_CFC_ (* Continuous Function Chart, elements in execution order *)
#0 WORD_TO_REAL(RD_2[0])
#1 DIV(#0, 100)
#2 SCHU_P2_1_M2_OBR <= #1
#3 dost_ton_2:TON(IN: NOT SCHU_P2_1_M2_OBR_ERROR, PT: t#10s)
#4 SR_DOST_M2:RS(SET: #3.Q, RESET1: SCHU_P2_1_M2_OBR_ERROR)
#5 fb_M2b30:ISTOK_GT(dost: #4.Q1, x: SCHU_P2_1_M2_OBR, ust: #14, shkal: -, gist: 1)
#6 SCHU_P2_1_M2_B30 <= #5.Xb
#7 fb_M2_OBRb45:ISTOK_GT(dost: #4.Q1, x: SCHU_P2_1_M2_OBR, ust: #16, shkal: -, gist: 1)
#8 SCHU_P2_1_M2_B45 <= #7.Xb
#9 fb_M2_OBRm0_1:ISTOK_LT(dost: #4.Q1, x: SCHU_P2_1_M2_OBR, ust: 0.1, shkal: -, gist: 1)
#10 SCHU_P2_1_M2_M0_1 <= #9.Xm
#11 fb_M2_OBRbSM:ISTOK_GT(dost: #4.Q1, x: SCHU_P2_1_M2_OBR, ust: SCHU_P2_1_M_MAXSPEED, shkal: -, gist: 1)
#12 SCHU_P2_1_M2_OBRBSM <= #11.Xb
(* 60% от частоты вращения *)
#13 DIV(SCHU_P2_1_M_MAXSPEED, 100)
#14 MUL(#13, 60)
#15 DIV(SCHU_P2_1_M_MAXSPEED, 100)
#16 MUL(#15, 85)
(* 85% от частоты вращения *)
_END_CFC_
END_PROGRAM

(* POU TZBiS/S/ALL_S, CFC *)
PROGRAM ALL_S
VAR
END_VAR
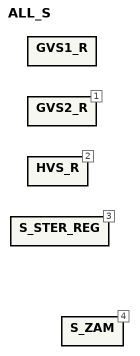
_CFC_ (* Continuous Function Chart, elements in execution order *)
#0 GVS1_R()
#1 GVS2_R()
#2 HVS_R()
#3 S_STER_REG()
#4 S_ZAM()
_END_CFC_
(* the same logic as Structured Text *)
GVS1_R();
GVS2_R();
HVS_R();
S_STER_REG();
S_ZAM();
END_PROGRAM

(* POU TZBiS/S/GVS1_R, CFC *)
PROGRAM GVS1_R
VAR
	rs_gvs1: RS;
	GVS1_RUN: BOOL;
END_VAR
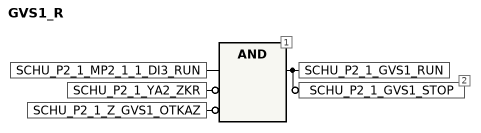
_CFC_ (* Continuous Function Chart, elements in execution order *)
#0 SCHU_P2_1_GVS1_RUN <= #1
#1 AND(SCHU_P2_1_MP2_1_1_DI3_RUN, NOT SCHU_P2_1_YA2_ZKR, NOT SCHU_P2_1_Z_GVS1_OTKAZ)
#2 SCHU_P2_1_GVS1_STOP <= NOT #1
_END_CFC_
END_PROGRAM

(* POU TZBiS/S/GVS2_R, CFC *)
PROGRAM GVS2_R
VAR
END_VAR
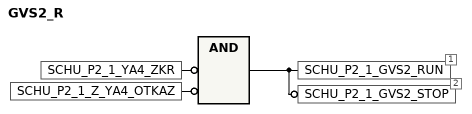
_CFC_ (* Continuous Function Chart, elements in execution order *)
#0 AND(NOT SCHU_P2_1_YA4_ZKR, NOT SCHU_P2_1_Z_YA4_OTKAZ)
#1 SCHU_P2_1_GVS2_RUN <= #0
#2 SCHU_P2_1_GVS2_STOP <= NOT #0
_END_CFC_
END_PROGRAM

(* POU TZBiS/S/HVS_R, CFC *)
PROGRAM HVS_R
VAR
END_VAR
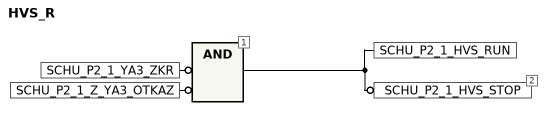
_CFC_ (* Continuous Function Chart, elements in execution order *)
#0 SCHU_P2_1_HVS_RUN <= #1
#1 AND(NOT SCHU_P2_1_YA3_ZKR, NOT SCHU_P2_1_Z_YA3_OTKAZ)
#2 SCHU_P2_1_HVS_STOP <= NOT #1
_END_CFC_
END_PROGRAM

(* POU TZBiS/S/S_STER_REG, CFC *)
PROGRAM S_STER_REG
VAR
	ZAD_S_Ster_Reg: TON;
END_VAR
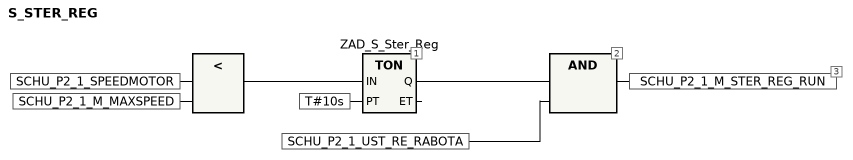
_CFC_ (* Continuous Function Chart, elements in execution order *)
#0 <(SCHU_P2_1_SPEEDMOTOR, SCHU_P2_1_M_MAXSPEED)
#1 ZAD_S_Ster_Reg:TON(IN: #0, PT: T#10s)
#2 AND(#1.Q, SCHU_P2_1_UST_RE_RABOTA)
#3 SCHU_P2_1_M_STER_REG_RUN <= #2
_END_CFC_
END_PROGRAM

(* POU TZBiS/S/S_ZAM, CFC *)
PROGRAM S_ZAM
VAR
	SR_ZAM: SR;
END_VAR
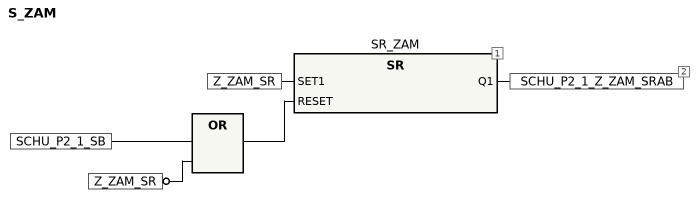
_CFC_ (* Continuous Function Chart, elements in execution order *)
#0 OR(SCHU_P2_1_SB, NOT Z_ZAM_SR)
#1 SR_ZAM:SR(SET1: Z_ZAM_SR, RESET: #0)
#2 SCHU_P2_1_Z_ZAM_SRAB <= #1.Q1
_END_CFC_
(* the same logic as Structured Text *)
SR_ZAM(SET1 := Z_ZAM_SR, RESET := SCHU_P2_1_SB OR NOT Z_ZAM_SR);
SCHU_P2_1_Z_ZAM_SRAB := SR_ZAM.Q1;
END_PROGRAM

(* POU TZBiS/TZB/ALL_TZB, CFC *)
PROGRAM ALL_TZB
VAR
END_VAR
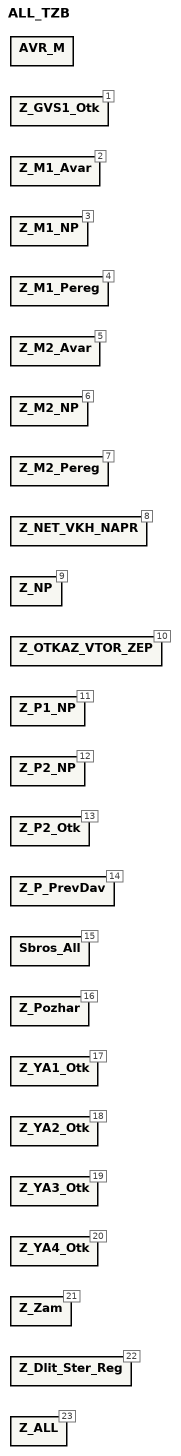
_CFC_ (* Continuous Function Chart, elements in execution order *)
#0 AVR_M()
#1 Z_GVS1_Otk()
#2 Z_M1_Avar()
#3 Z_M1_NP()
#4 Z_M1_Pereg()
#5 Z_M2_Avar()
#6 Z_M2_NP()
#7 Z_M2_Pereg()
#8 Z_NET_VKH_NAPR()
#9 Z_NP()
#10 Z_OTKAZ_VTOR_ZEP()
#11 Z_P1_NP()
#12 Z_P2_NP()
#13 Z_P2_Otk()
#14 Z_P_PrevDav()
#15 Sbros_All()
#16 Z_Pozhar()
#17 Z_YA1_Otk()
#18 Z_YA2_Otk()
#19 Z_YA3_Otk()
#20 Z_YA4_Otk()
#21 Z_Zam()
#22 Z_Dlit_Ster_Reg()
#23 Z_ALL()
_END_CFC_
(* the same logic as Structured Text *)
AVR_M();
Z_GVS1_Otk();
Z_M1_Avar();
Z_M1_NP();
Z_M1_Pereg();
Z_M2_Avar();
Z_M2_NP();
Z_M2_Pereg();
Z_NET_VKH_NAPR();
Z_NP();
Z_OTKAZ_VTOR_ZEP();
Z_P1_NP();
Z_P2_NP();
Z_P2_Otk();
Z_P_PrevDav();
Sbros_All();
Z_Pozhar();
Z_YA1_Otk();
Z_YA2_Otk();
Z_YA3_Otk();
Z_YA4_Otk();
Z_Zam();
Z_Dlit_Ster_Reg();
Z_ALL();
END_PROGRAM

(* POU TZBiS/TZB/AVR_M, CFC *)
PROGRAM AVR_M
VAR
	fb_HVACRC: FB_HVACRedundancyCtrl;
	RS_Pusk: RS;
	RT_Pusk: R_TRIG;


	rHours: ARRAY[1..8] OF REAL;
	uiCount: ARRAY[1..8] OF UINT;

	delayFBC: TIME := T#1s;
	overlap1Actuator: TIME := T#0s;
	maxOnLevel: UINT := 999;

	dtSystemTime: DT;
	fb_HVAC_GST: FB_HVACGetSystemTime;
	error: BOOL;
	RS_avr_kom: RS;
	RT_T: R_TRIG;
	TON_VKL: TON;
	TON_PUSK: TON;
	SCHU_P2_1_SA2_DI3_A: BOOL;
END_VAR
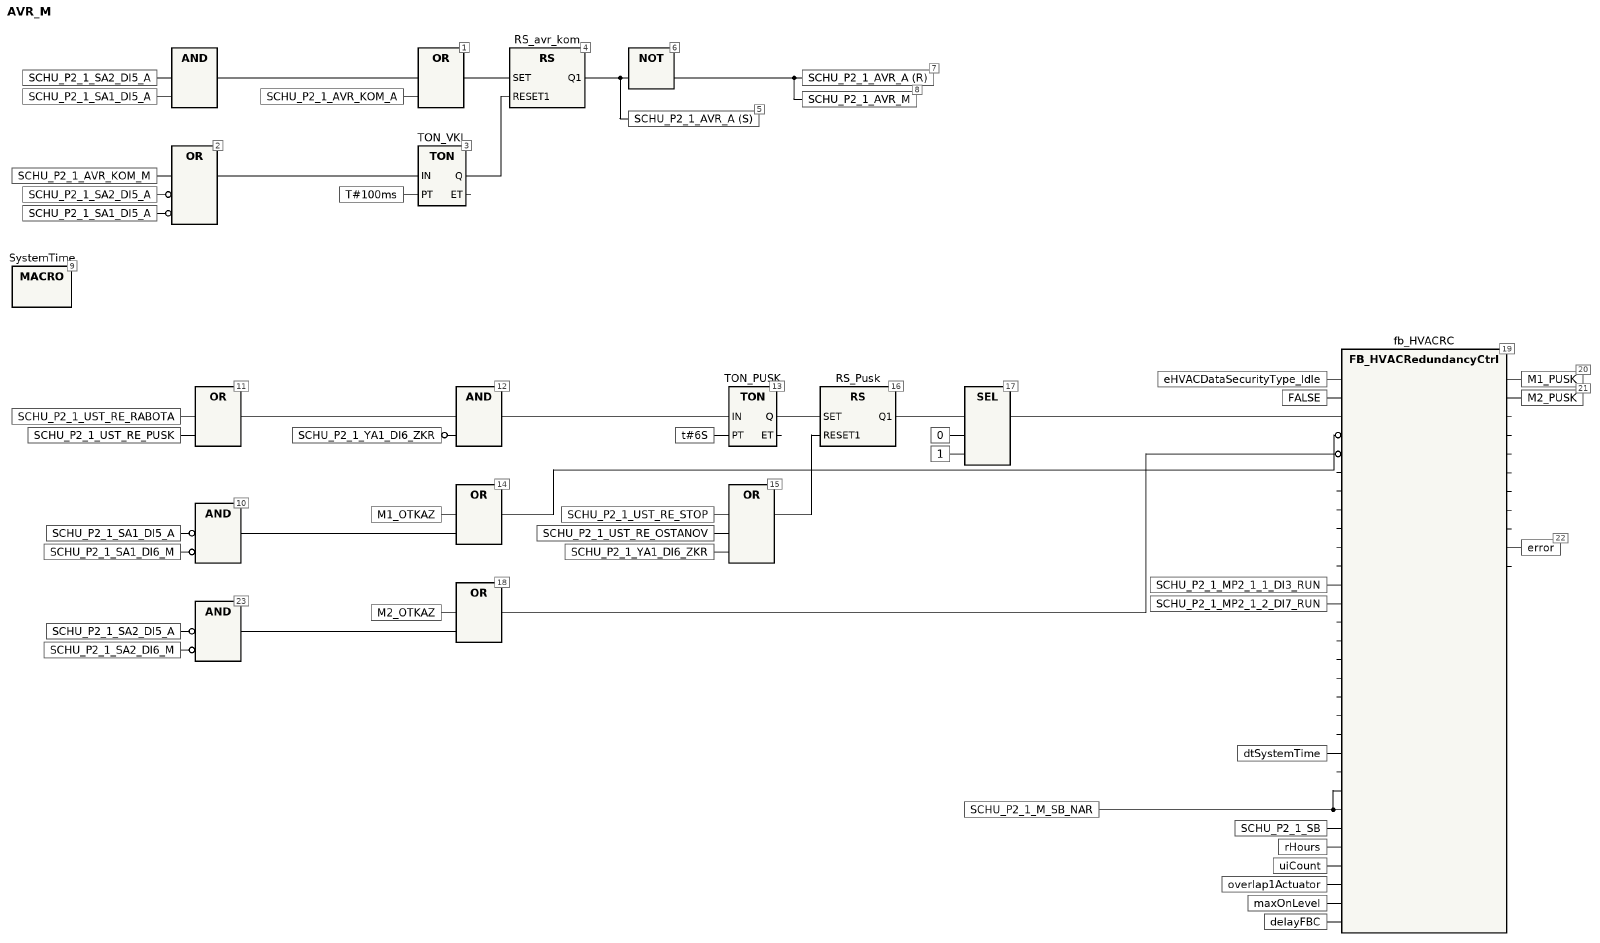
